FUNCTION_BLOCK FB_DEV_DigIn EXTENDS FB_DeviceBase IMPLEMENTS ITF_DigIn
VAR
	
END_VAR

{warning 'add property implementation'}
PROPERTY ActualValue : BOOL
GET
END_GET
SET
END_SET
END_PROPERTY

{warning 'add property implementation'}
PROPERTY FallingEdge : BOOL
GET
END_GET
SET
END_SET
END_PROPERTY

{warning 'add method implementation '}
METHOD FB_init : BOOL
VAR_INPUT
	(* if TRUE, the retain variables are initialized (warm start / cold start)*)
	bInitRetains	: BOOL;
	(* if TRUE, the instance afterwards gets moved into the copy code (online change)*)
	bInCopyCode	: BOOL;
END_VAR
END_METHOD

{warning 'add method implementation '}
METHOD Force : BOOL
VAR_INPUT
	ForceValue	: BOOL;
END_VAR
END_METHOD

{warning 'add method implementation '}
METHOD ResetForce : BOOL
END_METHOD

{warning 'add property implementation'}
PROPERTY RisingEdge : BOOL
GET
END_GET
SET
END_SET
END_PROPERTY

END_FUNCTION_BLOCK

(* stored: Version 1.1.0.1, ProductVersion 3.1.4024.12
   POU FB_DEV_DigIn: Id {bc7953ac-0b6f-4425-b2ef-ab2e018bf601}, SpecialFunc None
   Folder Methods: Id {13d3494c-b8c8-4e6e-b02d-eaa214c13190}
   Folder Properties: Id {ca254db0-bea6-43ee-b1f0-eae5b45aada0}
   Property ActualValue: Id {ad68ffcb-9a9b-4f28-b77f-1557373e8652}
   Get Get: Id {3bde900c-89d7-4d03-8deb-709b425cc65e}
   Set Set: Id {777b65e8-a2be-413d-b3f0-ec0a6f65a3b2}
   Property FallingEdge: Id {7df88f60-2daf-47fd-a2b4-6989ba2bf1c1}
   Get Get: Id {d30aaeee-c196-4bab-b959-5c3171b67cc9}
   Set Set: Id {01bd4f37-547f-4694-a243-f65da5e0ae5b}
   Method FB_init: Id {221f3045-662a-4918-999f-01d281278229}
   Method Force: Id {b36f677b-92fd-4909-9ef7-a239f577254a}
   Method ResetForce: Id {3c603f38-d38c-4363-a9a0-eb60af1221bc}
   Property RisingEdge: Id {107f28bb-cc6c-4af6-a990-dbccfb73e039}
   Get Get: Id {45aca2b1-8da5-445a-984f-e86e0b3855da}
   Set Set: Id {af15c501-7f40-40ef-9f66-e2cda7d2e16a} *)
